// TIA Portal V16 export
// export: Created 2024-12-03T15:41:41.0847655Z, ExportSetting WithDefaults, DisplayName Totally Integrated Automation Portal, DisplayVersion V16 Update 6, DisplayName TIA Portal Version Control Interface, DisplayVersion V16 Update 2, DisplayName TIA Portal Openness, DisplayVersion V16 Update 6, DisplayName TIA Portal Teamcenter Gateway, DisplayVersion V16, DisplayName SINAMICS Startdrive Advanced, DisplayVersion V16 Update 5, DisplayName SINAMICS Startdrive G130, G150, S120, S150, SINAMICS MV, S210, DisplayVersion V16 Update 5, DisplayName SINAMICS Startdrive G110M, G120, G120C, G120D, G120P, G115D, DisplayVersion V16 Update 5, DisplayName STEP 7 Professional, DisplayVersion V16 Update 6, DisplayName STEP 7 Safety, DisplayVersion V16, DisplayName WinCC Advanced / Unified PC, DisplayVersion V16 Update 6
FUNCTION_BLOCK "CycleRun"   // FB75, SCL
{ S7_Optimized_Access := 'TRUE' }
VERSION : 0.1
// stored: AutoNumber true, IsIECCheckEnabled false, IsRetainMemResEnabled false, MemoryReserve 100, SetENOAutomatically false, UDAEnableTagReadback false
   VAR_INPUT
      I_Start : Int := 1;
      I_End : Int := 10;
   END_VAR
   VAR_OUTPUT
      O_Cycle : Int;
   END_VAR
BEGIN
   #O_Cycle += 1;
   IF #O_Cycle > #I_End THEN
       #O_Cycle := #I_Start;
   END_IF;

   IF #O_Cycle < #I_Start THEN
       #O_Cycle := #I_Start;
   END_IF;
END_FUNCTION_BLOCK
